PROGRAM JIG003_NTG6
VAR
END_VAR

END_PROGRAM

(* stored: Version 1.1.0.1, ProductVersion 3.1.4022.18
   POU JIG003_NTG6: Id {3c51b419-1918-4961-a0f2-7ec3c0fba751}, SpecialFunc None *)
